FUNCTION_BLOCK FutureStatusLampControlCreator IMPLEMENTS InterfaceTaskCreator
VAR_INPUT
END_VAR
VAR_OUTPUT
END_VAR
VAR
	_ready_lamp : REFERENCE TO BOOL;
	_running_lamp : REFERENCE TO BOOL;
	_error_lamp : REFERENCE TO BOOL;
	_completed_lamp : REFERENCE TO BOOL;
	_lamp_state : UINT;
	_blink_interval : TIME := T#500MS;
END_VAR

METHOD create_future : InterfaceFuture
VAR_INPUT
    future_name : STRING;
END_VAR
VAR
    _p_future : POINTER TO FutureStatusLampControl;
END_VAR
_p_future := __NEW(FutureStatusLampControl);
_p_future^.future_name := future_name;

_p_future^.set_parameters(
    ready_lamp := _ready_lamp,
    running_lamp := _running_lamp,
    error_lamp := _error_lamp,
    completed_lamp := _completed_lamp,
    lamp_state := _lamp_state,
    blink_interval := _blink_interval
);

create_future := _p_future^;
END_METHOD

METHOD destroy_future : InterfaceFuture
VAR_INPUT
    future : InterfaceFuture;
END_VAR
VAR
    _p_future : POINTER TO FutureStatusLampControl;
END_VAR
IF __QUERYPOINTER(future, _p_future) THEN
	__DELETE(_p_future);
	IF _p_future = 0 THEN
		destroy_future := 0;
	END_IF
END_IF
END_METHOD

METHOD set_parameters : BOOL
VAR_INPUT
	ready_lamp : REFERENCE TO BOOL;
	running_lamp : REFERENCE TO BOOL;
	error_lamp : REFERENCE TO BOOL;
	completed_lamp : REFERENCE TO BOOL;
	lamp_state : UINT;
	blink_interval : TIME := T#500MS;
END_VAR
_ready_lamp REF= ready_lamp;
_running_lamp REF= running_lamp;
_error_lamp REF= error_lamp;
_completed_lamp REF= completed_lamp;
_lamp_state := lamp_state;
_blink_interval := blink_interval;
set_parameters := TRUE;
END_METHOD

END_FUNCTION_BLOCK

(* stored: Version 1.1.0.1, ProductVersion 3.1.4024.12
   POU FutureStatusLampControlCreator: Id {22222222-3333-4444-5555-666666666666}, SpecialFunc None
   Method create_future: Id {22222222-3333-4444-5555-777777777777}
   Method destroy_future: Id {22222222-3333-4444-5555-888888888888}
   Method set_parameters: Id {22222222-3333-4444-5555-999999999999} *)
